{attribute 'hide'}
{attribute clr [ExcludeFromApiDocumentation()]}
FUNCTION_BLOCK ABSTRACT TcoContextCompatibility EXTENDS TcoContext

{attribute 'hide'}
METHOD PROTECTED FINAL _Close
THIS^.Close();
END_METHOD

{attribute 'hide'}
METHOD PROTECTED FINAL _Open
THIS^.Open();
END_METHOD

END_FUNCTION_BLOCK

(* stored: Version 1.1.0.1
   POU TcoContextCompatibility: Id {13780382-a22f-0e35-3f52-856d3d4a5d71}, SpecialFunc None
   Method _Close: Id {ca63b2ce-d477-0f9f-02f9-549ed36e627f}
   Method _Open: Id {3cc7bb33-d3b0-01f7-3a73-00a2aa792610} *)
